FUNCTION_BLOCK FB_SK_StateManager

VAR
	bStartUpDone		: BOOL;	
	bFirstAbortDone		: BOOL;
	
	eCommand			: E_XMotion_Command;	
	eCommandOld			: E_XMotion_Command;
	eStatus				: E_XMotion_Status;	
	nCommandCounter		: UDINT;

END_VAR

METHOD PUBLIC Cycle
VAR_INPUT
END_VAR


	IF NOT bStartUpDone THEN					
		eStatus := E_XMotion_Status.StartUp;
	ELSIF NOT bFirstAbortDone THEN
		eStatus := E_XMotion_Status.Aborting;
	ELSE

		IF eCommand <> eCommandOld THEN
			eCommandOld := eCommand;
	
			nCommandCounter := nCommandCounter +1;
			
			
			CASE eCommand OF
				
			
			E_XMotion_Command.Abort:	
						eStatus := E_XMotion_Status.Aborting;	
			
			E_XMotion_Command.Reset:
						IF eStatus = E_XMotion_Status.Aborted THEN
							eStatus := E_XMotion_Status.Resetting;	
						END_IF
				
			E_XMotion_Command.Prepare:
						IF eStatus = E_XMotion_Status.Stopped THEN
							eStatus := E_XMotion_Status.Preparing;	
						END_IF	
			
			E_XMotion_Command.Start:
						IF eStatus = E_XMotion_Status.Prepared THEN
							eStatus := E_XMotion_Status.Execute;	
						END_IF	

			E_XMotion_Command.HoldOnError:
						eStatus := E_XMotion_Status.HoldOnError;

					
			END_CASE
		END_IF
		
	END_IF
END_METHOD

METHOD PUBLIC StateComplete : BOOL
VAR_INPUT
END_VAR




	CASE eStatus OF
		
	E_XMotion_Status.StartUp:
				bStartUpDone := TRUE;
				
	E_XMotion_Status.Aborting:
				bFirstAbortDone := TRUE;	
				eStatus := E_XMotion_Status.Aborted;	
	
	E_XMotion_Status.Resetting:
				eStatus := E_XMotion_Status.Stopped;
		
	E_XMotion_Status.Preparing:
				eStatus := E_XMotion_Status.Prepared;
	
				
	END_CASE
END_METHOD

PROPERTY Status : E_XMotion_Status
GET
Status := eStatus;
END_GET
END_PROPERTY

PROPERTY XMotionCommand : E_XMotion_Command
SET
eCommand := XMotionCommand;
END_SET
END_PROPERTY

END_FUNCTION_BLOCK

(* stored: Version 1.1.0.1, ProductVersion 3.1.4024.9
   POU FB_SK_StateManager: Id {ba6ea3a9-f4d6-452f-bbd4-8f581c1dd188}, SpecialFunc None
   Method Cycle: Id {2b480e1d-388a-4266-9461-4240b3740607}
   Method StateComplete: Id {bb432478-cdb4-46c1-ae1e-3b9c78e8a7c5}
   Property Status: Id {cd3b1284-33bd-4147-894f-f84c692ae866}
   Get Get: Id {7cc5837d-c26d-4941-86af-4b977c7f86dd}
   Property XMotionCommand: Id {b194e988-2fd8-448f-985b-c21173801e09}
   Set Set: Id {5bed3948-1fe7-419e-9df8-105a5a39f66c} *)
